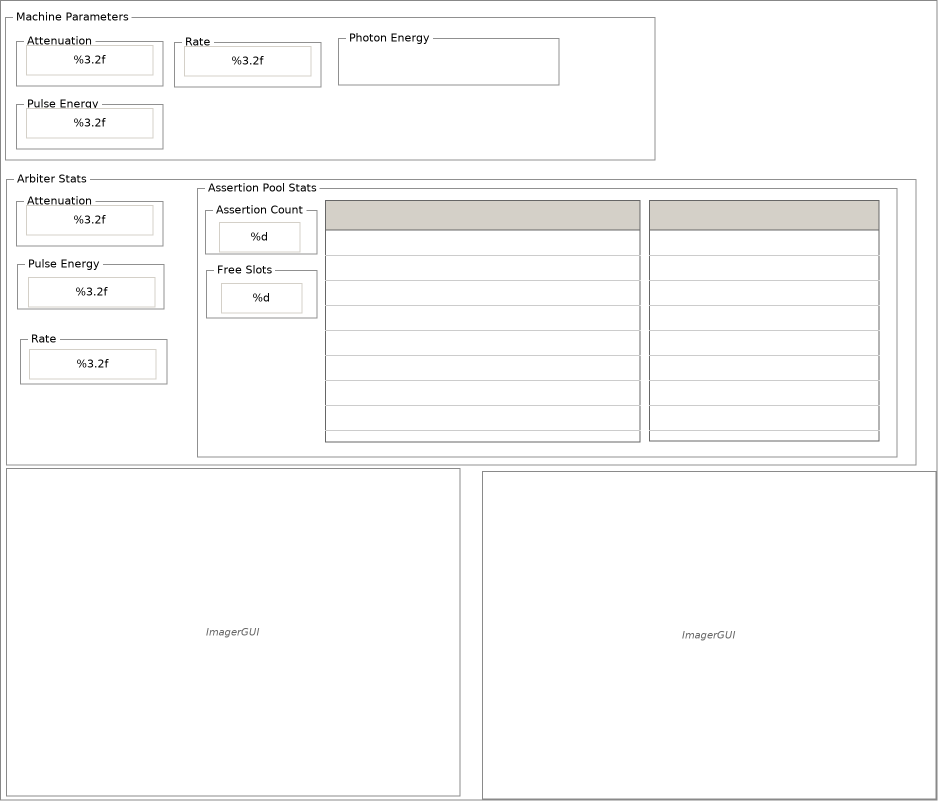
VISUALIZATION Visualization  // 938x801
    GroupBox (5,9 650x151), "Machine Parameters"
        GroupBox (11,24 147x53), "Attenuation"
            Textfield (10,12 127x30), "%3.2f", text variable: PMPS_GVL_BeamParams.stCurrentBeamParameters.fAtt
        GroupBox (11,87 147x53), "Pulse Energy"
            Textfield (10,12 127x30), "%3.2f", text variable: PMPS_GVL_BeamParams.stCurrentBeamParameters.fPP_mJ
        GroupBox (169,25 147x53), "Rate"
            Textfield (10,12 127x30), "%3.2f", text variable: PMPS_GVL_BeamParams.stCurrentBeamParameters.nRate
        GroupBox (333,21 221x55), "Photon Energy"
    GroupBox (6,171 910x294), "Arbiter Stats"
        GroupBox (191,9 700x277), "Assertion Pool Stats"
            GroupBox (9,82 111x56), "Free Slots"
                Textfield (15,21 81x30), "%d", text variable: fbArbiter.fbBPAssertionPool.hTable.nFree
            GroupBox (8,22 112x52), "Assertion Count"
                Textfield (14,20 81x30), "%d", text variable: fbArbiter.fbBPAssertionPool.hTable.nCount
            Table (128,20 315x242), data array: fbArbiter.fbBPAssertionPool.dataPool
                p3854506369: fbArbiter.fbBPAssertionPool.dataPool[INDEX].fAtt
                p1892666644: fbArbiter.fbBPAssertionPool.dataPool[INDEX].fPP_mJ
                p338671338: fbArbiter.fbBPAssertionPool.dataPool[INDEX].fUpper_eV
                p2170511999: fbArbiter.fbBPAssertionPool.dataPool[INDEX].fLower_eV
                p1755163831: Upper eV
                p4092479075: Lower eV
            Table (452,20 230x241), data array: fbArbiter.fbBPAssertionPool.entries
                p3854506369: fbArbiter.fbBPAssertionPool.entries[INDEX].key
                p1892666644: fbArbiter.fbBPAssertionPool.entries[INDEX].value
                p338671338: fbArbiter.fbBPAssertionPool.entries[INDEX].lock
                p2170511999: fbArbiter.fbBPAssertionPool.entries[INDEX].pNext
                p3723444502: fbArbiter.fbBPAssertionPool.entries[INDEX].pNextFree
                p1218418051: fbArbiter.fbBPAssertionPool.entries[INDEX].pNextGlob
                p2232123230: Assertion ID
        GroupBox (10,22 147x53), "Attenuation"
            Textfield (10,12 127x30), "%3.2f", text variable: fbArbiter.q_stBeamParams.fAtt
        GroupBox (11,85 147x53), "Pulse Energy"
            Textfield (11,21 127x30), "%3.2f", text variable: fbArbiter.q_stBeamParams.fPP_mJ
        GroupBox (14,160 147x53), "Rate"
            Textfield (9,18 127x30), "%3.2f", text variable: fbArbiter.stOutputBP.nRate
    Frame (6,468 454x328)
        shows ImagerGUI(stDevice := MAIN.fbDev1.stDevice)
    Frame (482,471 454x328)
        shows ImagerGUI(stDevice := MAIN.fbDev2.stDevice)
END_VISUALIZATION

(* stored: Version 1.1.0.1, ProductVersion 3.1.4022.18
   Visu Visualization: Id {e2d11be7-f40a-0a2a-160a-0d1b47b9df45} *)
